{attribute 'pack_mode' := '2'}
TYPE U_XTS_TRANSPORT_STATE :
UNION
  stState             : ST_XTS_TRANSPORT_STATE;
  byState   AT %i*    : ARRAY[1..SIZEOF(ST_XTS_TRANSPORT_STATE)] OF BYTE;
END_UNION
END_TYPE

(* stored: Version 1.1.0.1
   DUT U_XTS_TRANSPORT_STATE: Id {52bb505b-c786-462c-8e59-10e2be0c71c5} *)
